Staubli VAL3: setWordAt.pgx

public program setWordAt(num x_nByteIndex, num x_nWord, num& x_nBuffer[])
  local string l_sBinWord
  local num l_nLOword
  local num l_nHIword
  local string l_sTempBinByte
begin

  //gestione del segno???
  if x_nWord<0 or x_nWord>power(2,16)-1
    x_nBuffer[x_nByteIndex] = 0
    x_nBuffer[x_nByteIndex+1] = 0
    return
  endIf

  l_sBinWord=""
  call bitOp:BitWord(x_nWord, l_sBinWord)
  call bitOp:shiftRight(l_sBinWord, 8)
  call bitOp:BinToDec(l_sBinWord, l_nLOword)

  l_sBinWord=""
  call bitOp:BitWord(x_nWord, l_sBinWord)
  call bitOp:boolAnd(l_sBinWord, "0000000011111111", l_sTempBinByte)
  call bitOp:BinToDec(l_sTempBinByte, l_nHIword)

  x_nBuffer[x_nByteIndex] = l_nLOword
  x_nBuffer[x_nByteIndex+1] = l_nHIword

end
